(* Logix 5000 project; controller cal1632 1756-L62 rev 16.20; software revision 16.05; part 7 of 61 *)
(* tags used below, declared in another part *)
   tmrFlash : TIMER[4];   // Flash Timer
   aaa_aaa_temp : BOOL;
   FAULT : BOOL;
   FlashBit_500MSec : BOOL;   // Flash Bit 500 MSec
   p00_FlashBit_1Sec : BOOL;   // System Flash Bit 1 Second
   p00_wac : Accumulator;   // Winder Accumulator
   p01_int_from_oxidizer : INT[10];
   p01_param_master_accel : REAL;
   p01_param_master_decel : REAL;
   p01_param_master_jog_accel : REAL;
   p01_param_master_jog_decel : REAL;
   p01_param_master_jog_speed : REAL;
   p01_param_oven_timer_presets : DINT[32];
   p01_param_slow_speed_sp : REAL;
   p01_param_start_delay : REAL;
   p01_param_tension_deviation : REAL;
   p01_recipe_active : recipe;
   p01r01 : routine;
   p01r02_do_buzzer : BOOL;
   p01r02_do_buzzer_LINE : BOOL;
   p01r02_do_green_stack_light_lel : BOOL;
   p01r02_do_green_stack_light_LINE : BOOL;
   p01r02_do_horn : BOOL;
   p01r02_do_red_stack_light : BOOL;
   p01r02_do_red_stack_light_LINE : BOOL;
   p01r02_do_yellow_stack_light : BOOL;
   p01r02_do_yellow_stack_light_LINE : BOOL;
   p01r02_plc_scan_time_in_sec : REAL;
   p01r02_timer_second : TIMER[2];
   p01r09 : routine;
   p01r09_mode_run : BOOL;
   p01r09_open_oven : BOOL;
   p01r09_pb_global_reset : BOOL;
   p01r09_pb_line_jog : BOOL;
   p01r09_request_line_jog : BOOL;
   p01r10 : routine;
   p01r10_timer_fault : TIMER[4];
   p01r10_timer_warning : TIMER[4];
   p01r10_unack_fault_ex : BOOL;
   p01r10_unack_warn_ex : BOOL;
   p01r11 : routine;
   p01r11_timer_fault : TIMER[4];
   p01r11_timer_warning : TIMER[4];
   p01r12 : routine;
   p01r12_accel_rate : REAL;
   p01r12_decel_rate : REAL;
   p01r12_line_at_speed : BOOL;
   p01r12_master_acel_decel_ramp : SYS_ACC_DEC_RAMP;
   p01r12_master_ramped_speed : REAL;
   p01r12_ramped_setpoint : REAL;
   p01r12_request_any_jog_thread : BOOL;
   p01r12_selected_line_speed : REAL;
   p01r12_timer_fault : TIMER[8];
   p01r12_timer_warning : TIMER[8];
   p01r12_zero_line_speed : BOOL;
   p01r13 : routine;
   p01r13_check_status : BOOL;
   p01r13_check_status_time : REAL;
   p01r13_check_status_timer : TIMER;
   p01r13_check_tension : TIMER;
   p01r13_letoff_tension_ok : BOOL;
   p01r13_LFL_stop : BOOL;
   p01r13_line_running : BOOL;
   p01r13_line_slow_ramp : BOOL;
   p01r13_line_start : SYS_ENC;
   p01r13_oven_temp_ok : BOOL;
   p01r13_pb_start : BOOL;
   p01r13_pb_stop : BOOL;
   p01r13_permissive_drives : BOOL;
   p01r13_permissive_line_run : BOOL;
   p01r13_permissive_oven : BOOL;
   p01r13_permissive_oxidizer : BOOL;
   p01r13_request_run : BOOL;
   p01r13_request_stop : BOOL;
   p01r13_state : DINT;
   p01r13_status : DINT;
   p01r13_system_mode_run : BOOL;
   p01r13_temperature_status_check : TIMER;
   p01r13_tension_ok : BOOL;
   p01r13_timer_line_start_warning_dwell : TIMER;
   p01r13_timer_line_stop_dwell : TIMER;
   p01r13_timer_switch_to_stretch_dwell : TIMER;
   p01r13_ts1_tension_ok : BOOL;
   p01r13_ts2_tension_ok : BOOL;
   p01r13_winder_tension_ok : BOOL;
   p01r14 : routine;
   p02_dint_from_hmi : hmi_dint;
   p02_real_from_hmi : hmi_real;
   p11r30 : routine;
   p11r30_request_heat : BOOL;
   p11r31 : routine;
   p12r30 : routine;
   p12r30_request_heat : BOOL;
   p12r31 : routine;
   p13r30 : routine;
   p13r30_request_cool : BOOL;
   p20_di_acc_empty : BOOL;
   p20_do_close_nip : BOOL;
   p20r02_letoff_selection_dwell : TIMER;
   p20r10 : routine;
   p20r10_pid_tens : PID;
   p20r15 : routine;
   p20r15_loa_on : BOOL;
   p20r16 : routine;
   p20r16_lob_on : BOOL;
   p20r18_index_complete : BOOL;
   p22_param_ts1_jog_speed : REAL;
   p22r09_mode_run : BOOL;
   p22r09_mode_thread : BOOL;
   p22r09_pb_jog_fwd : BOOL;
   p22r09_pb_jog_rev : BOOL;
   p22r10_pid_psn : PID;
   p22r11 : routine;
   p22r11_request_thread_fwd : BOOL;
   p22r11_request_thread_rev : BOOL;
   p23_di_impreg_tank_up : BOOL;
   p23_param_mtr_jog_speed : REAL;
   p23r02 : routine;
   p23r15 : routine;
   p25_param_ts2_jog_speed : REAL;
   p25r09_mode_run : BOOL;
   p25r09_mode_thread : BOOL;
   p25r09_pb_jog_fwd : BOOL;
   p25r09_pb_jog_rev : BOOL;
   p25r10_pid_psn : PID;
   p25r11 : routine;
   p25r11_request_thread_fwd : BOOL;
   p25r11_request_thread_rev : BOOL;
   p28r11 : routine;
   p29_param_winder_jog_speed : REAL;
   p29r02_winder_selection_dwell : TIMER;
   p29r10_tension_error : REAL;   // Winder Winder A Tension Error winder_tension_sp - Load Cell [lbf]
   p29r11_line_start : BOOL;
   p29r11_line_stop : BOOL;
   p29r15 : routine;
   p29r15_wdra_active : BOOL;
   p29r16 : routine;
   p29r16_wdrb_active : BOOL;
   p31r09 : routine;
(* P01_System, continued *)

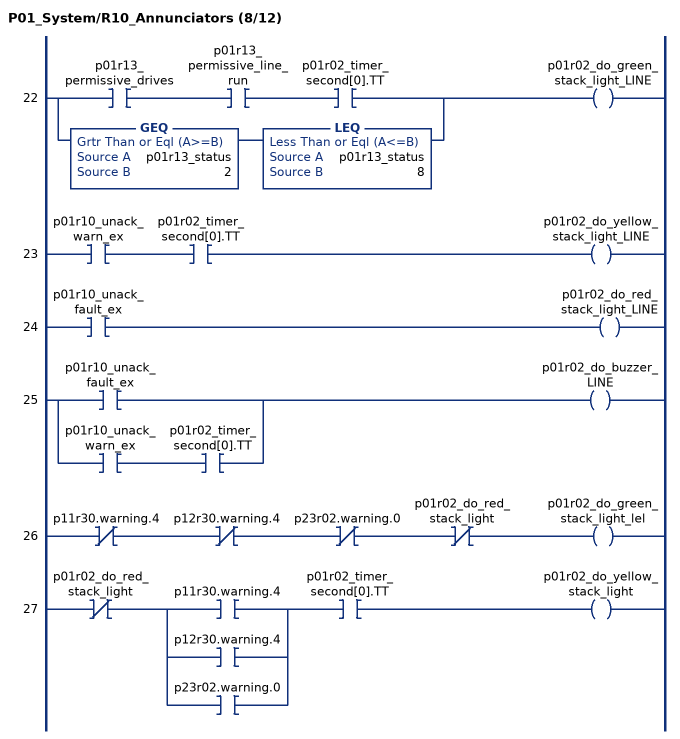
   [picture p99: P01_System/R10_Annunciators rungs 22-27]
   22: [XIC(p01r13_permissive_drives) XIC(p01r13_permissive_line_run) XIC(p01r02_timer_second[0].TT) ,GEQ(p01r13_status,2) LEQ(p01r13_status,8) ]OTE(p01r02_do_green_stack_light_LINE);
   23: XIC(p01r10_unack_warn_ex)XIC(p01r02_timer_second[0].TT)OTE(p01r02_do_yellow_stack_light_LINE);
   24: XIC(p01r10_unack_fault_ex)OTE(p01r02_do_red_stack_light_LINE);
   25: [XIC(p01r10_unack_fault_ex) ,XIC(p01r10_unack_warn_ex) XIC(p01r02_timer_second[0].TT) ]OTE(p01r02_do_buzzer_LINE);
   26: XIO(p11r30.warning.4)XIO(p12r30.warning.4)XIO(p23r02.warning.0)XIO(p01r02_do_red_stack_light)OTE(p01r02_do_green_stack_light_lel);
   27: XIO(p01r02_do_red_stack_light)[XIC(p11r30.warning.4) ,XIC(p12r30.warning.4) ,XIC(p23r02.warning.0) ]XIC(p01r02_timer_second[0].TT)OTE(p01r02_do_yellow_stack_light);
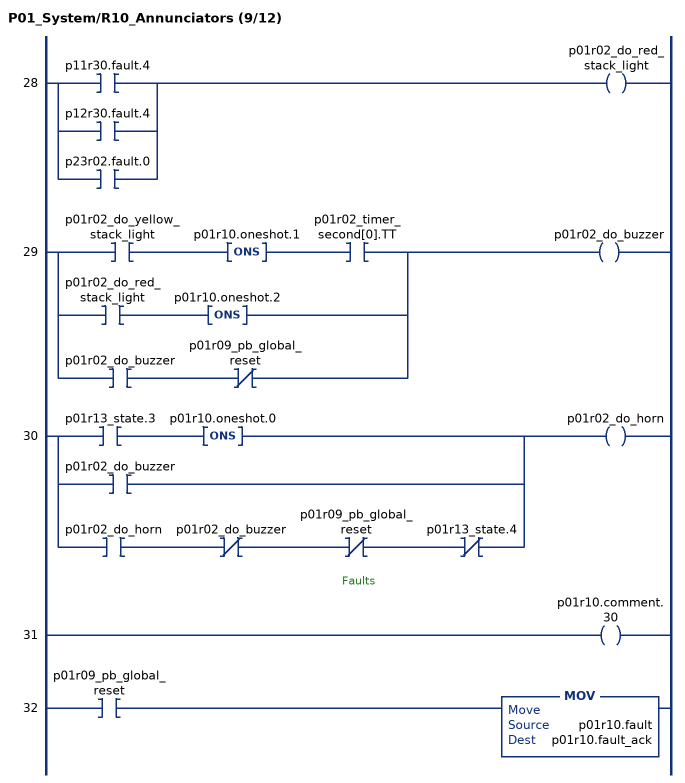
   28: [XIC(p11r30.fault.4) ,XIC(p12r30.fault.4) ,XIC(p23r02.fault.0) ]OTE(p01r02_do_red_stack_light);
   29: [[XIC(p01r02_do_yellow_stack_light) ONS(p01r10.oneshot.1) XIC(p01r02_timer_second[0].TT) ,XIC(p01r02_do_red_stack_light) ONS(p01r10.oneshot.2) ] ,XIC(p01r02_do_buzzer) XIO(p01r09_pb_global_reset) ]OTE(p01r02_do_buzzer);
   30: [[XIC(p01r13_state.3) ONS(p01r10.oneshot.0) ,XIC(p01r02_do_buzzer) ] ,XIC(p01r02_do_horn) XIO(p01r02_do_buzzer) XIO(p01r09_pb_global_reset) XIO(p01r13_state.4) ]OTE(p01r02_do_horn);
   // Faults
   31: OTE(p01r10.comment.30);
   32: XIC(p01r09_pb_global_reset)MOV(p01r10.fault,p01r10.fault_ack);
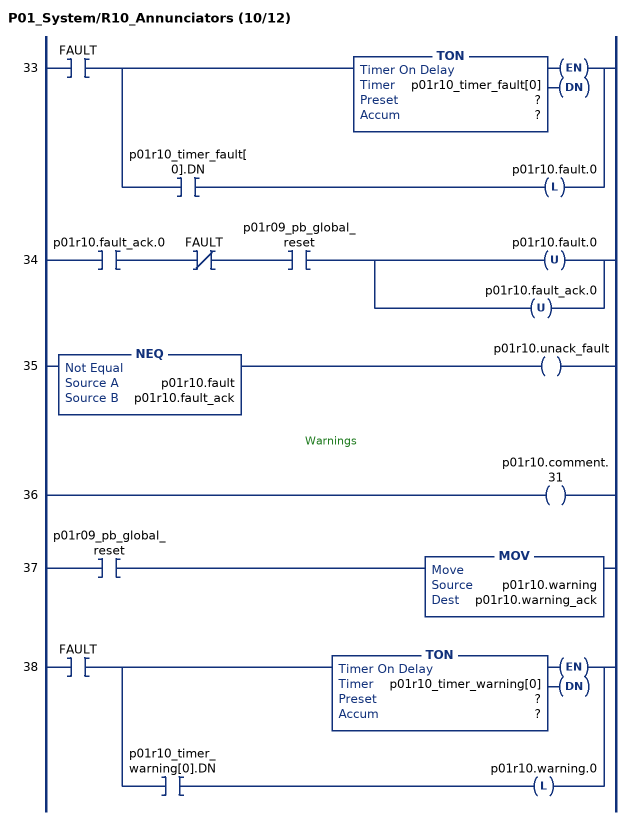
   33: XIC(FAULT)[TON(p01r10_timer_fault[0],?,?) ,XIC(p01r10_timer_fault[0].DN) OTL(p01r10.fault.0) ];
   34: XIC(p01r10.fault_ack.0)XIO(FAULT)XIC(p01r09_pb_global_reset)[OTU(p01r10.fault.0) ,OTU(p01r10.fault_ack.0) ];
   35: NEQ(p01r10.fault,p01r10.fault_ack)OTE(p01r10.unack_fault);
   // Warnings
   36: OTE(p01r10.comment.31);
   37: XIC(p01r09_pb_global_reset)MOV(p01r10.warning,p01r10.warning_ack);
   38: XIC(FAULT)[TON(p01r10_timer_warning[0],?,?) ,XIC(p01r10_timer_warning[0].DN) OTL(p01r10.warning.0) ];
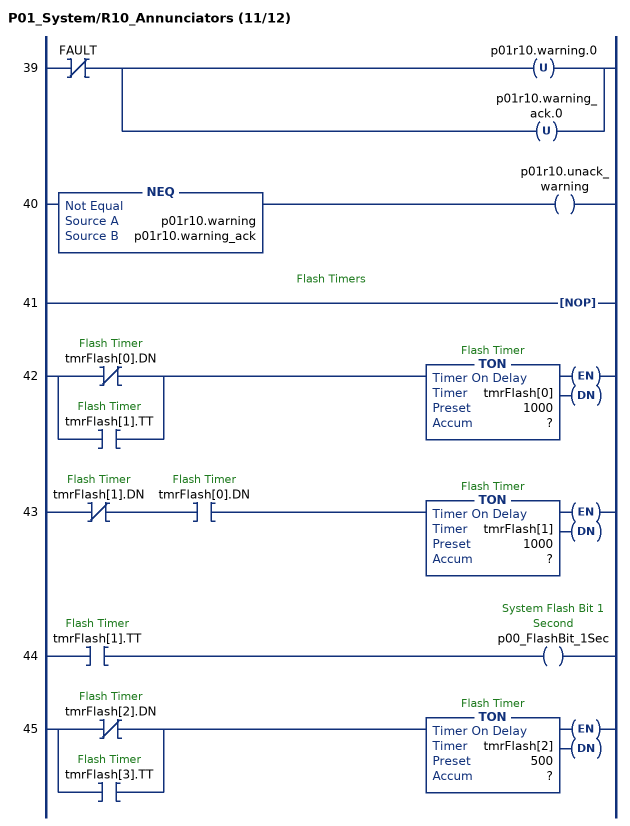
   39: XIO(FAULT)[OTU(p01r10.warning.0) ,OTU(p01r10.warning_ack.0) ];
   40: NEQ(p01r10.warning,p01r10.warning_ack)OTE(p01r10.unack_warning);
   // Flash Timers
   41: NOP();
   42: [XIO(tmrFlash[0].DN) ,XIC(tmrFlash[1].TT) ]TON(tmrFlash[0],?,?);
   43: XIO(tmrFlash[1].DN)XIC(tmrFlash[0].DN)TON(tmrFlash[1],?,?);
   44: XIC(tmrFlash[1].TT)OTE(p00_FlashBit_1Sec);
   45: [XIO(tmrFlash[2].DN) ,XIC(tmrFlash[3].TT) ]TON(tmrFlash[2],?,?);
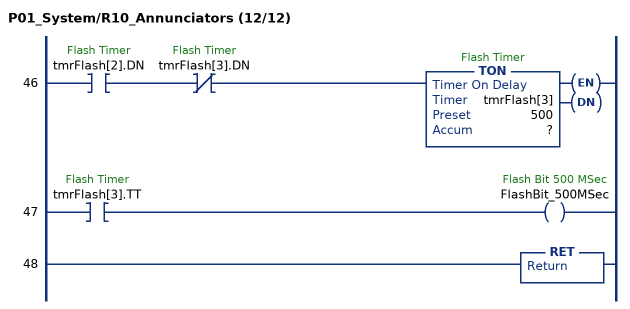
   46: XIC(tmrFlash[2].DN)XIO(tmrFlash[3].DN)TON(tmrFlash[3],?,?);
   47: XIC(tmrFlash[3].TT)OTE(FlashBit_500MSec);
   48: RET();
END_ROUTINE

ROUTINE R11_Oven_Timer_Presets   (* ladder *)
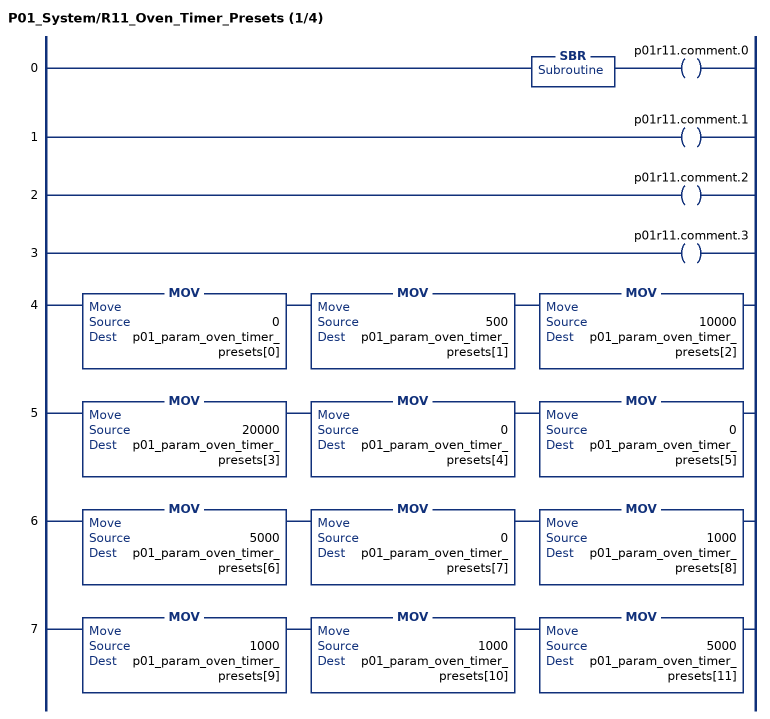
   0: SBR()OTE(p01r11.comment.0);
   1: OTE(p01r11.comment.1);
   2: OTE(p01r11.comment.2);
   3: OTE(p01r11.comment.3);
   4: MOV(0,p01_param_oven_timer_presets[0])MOV(500,p01_param_oven_timer_presets[1])MOV(10000,p01_param_oven_timer_presets[2]);
   5: MOV(20000,p01_param_oven_timer_presets[3])MOV(0,p01_param_oven_timer_presets[4])MOV(0,p01_param_oven_timer_presets[5]);
   6: MOV(5000,p01_param_oven_timer_presets[6])MOV(0,p01_param_oven_timer_presets[7])MOV(1000,p01_param_oven_timer_presets[8]);
   7: MOV(1000,p01_param_oven_timer_presets[9])MOV(1000,p01_param_oven_timer_presets[10])MOV(5000,p01_param_oven_timer_presets[11]);
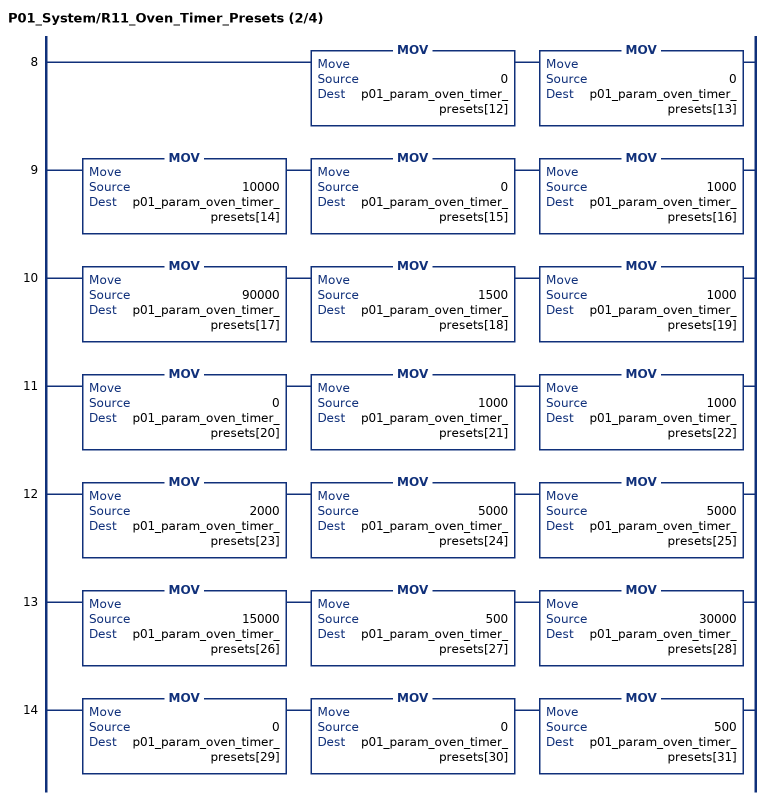
   8: MOV(0,p01_param_oven_timer_presets[12])MOV(0,p01_param_oven_timer_presets[13]);
   9: MOV(10000,p01_param_oven_timer_presets[14])MOV(0,p01_param_oven_timer_presets[15])MOV(1000,p01_param_oven_timer_presets[16]);
   10: MOV(90000,p01_param_oven_timer_presets[17])MOV(1500,p01_param_oven_timer_presets[18])MOV(1000,p01_param_oven_timer_presets[19]);
   11: MOV(0,p01_param_oven_timer_presets[20])MOV(1000,p01_param_oven_timer_presets[21])MOV(1000,p01_param_oven_timer_presets[22]);
   12: MOV(2000,p01_param_oven_timer_presets[23])MOV(5000,p01_param_oven_timer_presets[24])MOV(5000,p01_param_oven_timer_presets[25]);
   13: MOV(15000,p01_param_oven_timer_presets[26])MOV(500,p01_param_oven_timer_presets[27])MOV(30000,p01_param_oven_timer_presets[28]);
   14: MOV(0,p01_param_oven_timer_presets[29])MOV(0,p01_param_oven_timer_presets[30])MOV(500,p01_param_oven_timer_presets[31]);
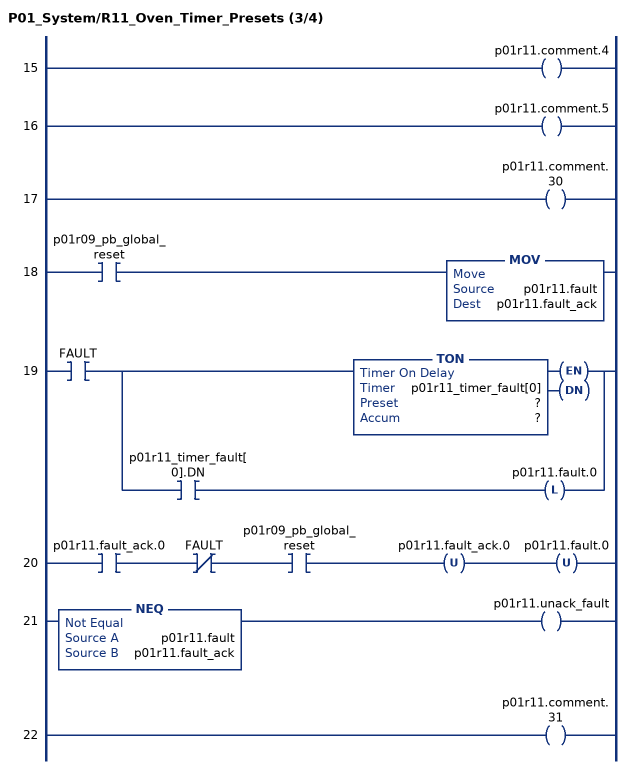
   15: OTE(p01r11.comment.4);
   16: OTE(p01r11.comment.5);
   17: OTE(p01r11.comment.30);
   18: XIC(p01r09_pb_global_reset)MOV(p01r11.fault,p01r11.fault_ack);
   19: XIC(FAULT)[TON(p01r11_timer_fault[0],?,?) ,XIC(p01r11_timer_fault[0].DN) OTL(p01r11.fault.0) ];
   20: XIC(p01r11.fault_ack.0)XIO(FAULT)XIC(p01r09_pb_global_reset)OTU(p01r11.fault_ack.0)OTU(p01r11.fault.0);
   21: NEQ(p01r11.fault,p01r11.fault_ack)OTE(p01r11.unack_fault);
   22: OTE(p01r11.comment.31);
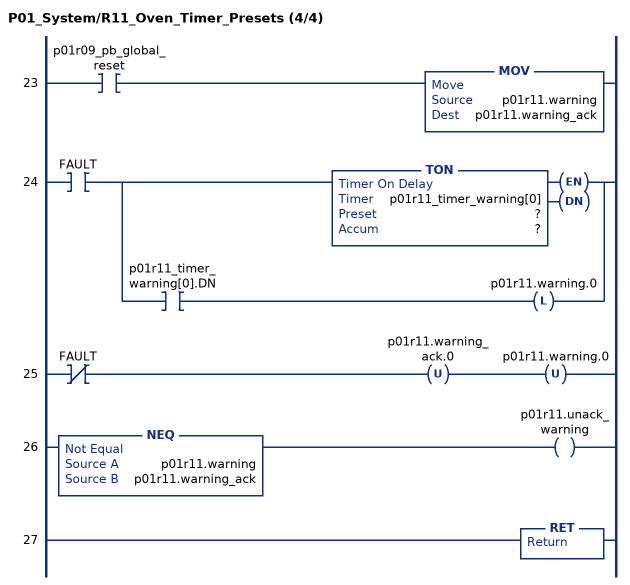
   23: XIC(p01r09_pb_global_reset)MOV(p01r11.warning,p01r11.warning_ack);
   24: XIC(FAULT)[TON(p01r11_timer_warning[0],?,?) ,XIC(p01r11_timer_warning[0].DN) OTL(p01r11.warning.0) ];
   25: XIO(FAULT)OTU(p01r11.warning_ack.0)OTU(p01r11.warning.0);
   26: NEQ(p01r11.warning,p01r11.warning_ack)OTE(p01r11.unack_warning);
   27: RET();
END_ROUTINE

ROUTINE R12_Line_Accel_Decel_Control   (* ladder *)
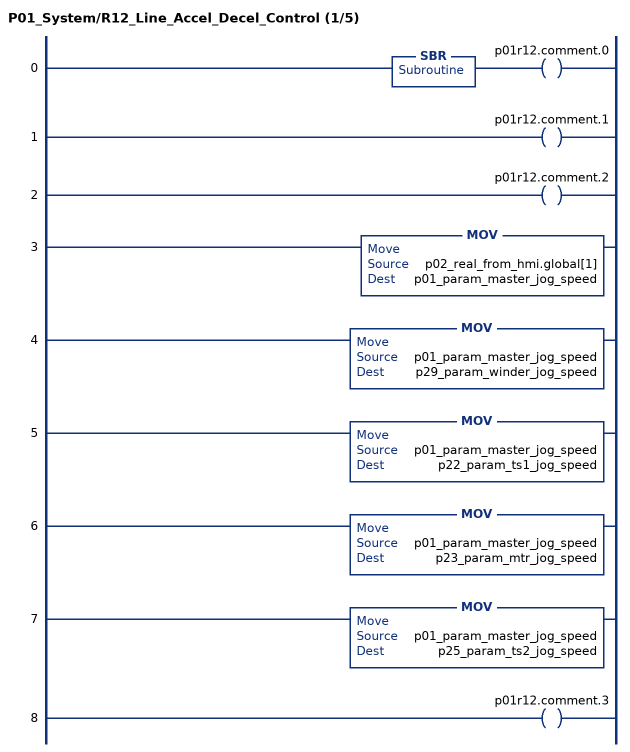
   0: SBR()OTE(p01r12.comment.0);
   1: OTE(p01r12.comment.1);
   2: OTE(p01r12.comment.2);
   3: MOV(p02_real_from_hmi.global[1],p01_param_master_jog_speed);
   4: MOV(p01_param_master_jog_speed,p29_param_winder_jog_speed);
   5: MOV(p01_param_master_jog_speed,p22_param_ts1_jog_speed);
   6: MOV(p01_param_master_jog_speed,p23_param_mtr_jog_speed);
   7: MOV(p01_param_master_jog_speed,p25_param_ts2_jog_speed);
   8: OTE(p01r12.comment.3);
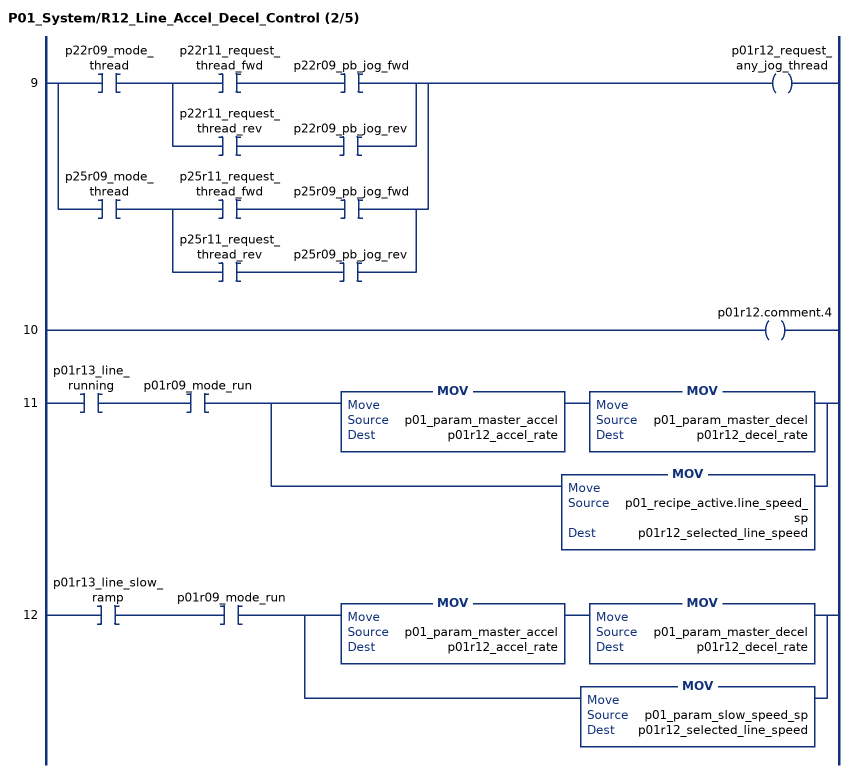
   9: [XIC(p22r09_mode_thread) [XIC(p22r11_request_thread_fwd) XIC(p22r09_pb_jog_fwd) ,XIC(p22r11_request_thread_rev) XIC(p22r09_pb_jog_rev) ] ,XIC(p25r09_mode_thread) [XIC(p25r11_request_thread_fwd) XIC(p25r09_pb_jog_fwd) ,XIC(p25r11_request_thread_rev) XIC(p25r09_pb_jog_rev) ] ]OTE(p01r12_request_any_jog_thread);
   10: OTE(p01r12.comment.4);
   11: XIC(p01r13_line_running)XIC(p01r09_mode_run)[MOV(p01_param_master_accel,p01r12_accel_rate) MOV(p01_param_master_decel,p01r12_decel_rate) ,MOV(p01_recipe_active.line_speed_sp,p01r12_selected_line_speed) ];
   12: XIC(p01r13_line_slow_ramp)XIC(p01r09_mode_run)[MOV(p01_param_master_accel,p01r12_accel_rate) MOV(p01_param_master_decel,p01r12_decel_rate) ,MOV(p01_param_slow_speed_sp,p01r12_selected_line_speed) ];
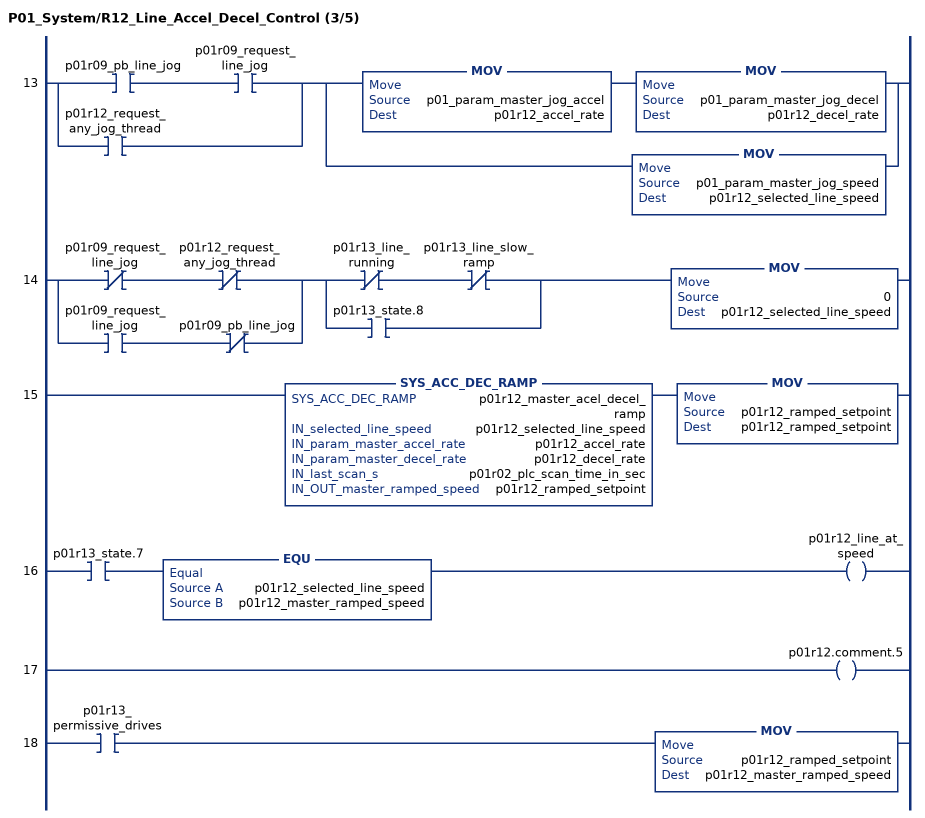
   13: [XIC(p01r09_pb_line_jog) XIC(p01r09_request_line_jog) ,XIC(p01r12_request_any_jog_thread) ][MOV(p01_param_master_jog_accel,p01r12_accel_rate) MOV(p01_param_master_jog_decel,p01r12_decel_rate) ,MOV(p01_param_master_jog_speed,p01r12_selected_line_speed) ];
   14: [XIO(p01r09_request_line_jog) XIO(p01r12_request_any_jog_thread) ,XIC(p01r09_request_line_jog) XIO(p01r09_pb_line_jog) ][XIO(p01r13_line_running) XIO(p01r13_line_slow_ramp) ,XIC(p01r13_state.8) ]MOV(0,p01r12_selected_line_speed);
   15: SYS_ACC_DEC_RAMP(p01r12_master_acel_decel_ramp,p01r12_selected_line_speed,p01r12_accel_rate,p01r12_decel_rate,p01r02_plc_scan_time_in_sec,p01r12_ramped_setpoint)MOV(p01r12_ramped_setpoint,p01r12_ramped_setpoint);
   16: XIC(p01r13_state.7)EQU(p01r12_selected_line_speed,p01r12_master_ramped_speed)OTE(p01r12_line_at_speed);
   17: OTE(p01r12.comment.5);
   18: XIC(p01r13_permissive_drives)MOV(p01r12_ramped_setpoint,p01r12_master_ramped_speed);
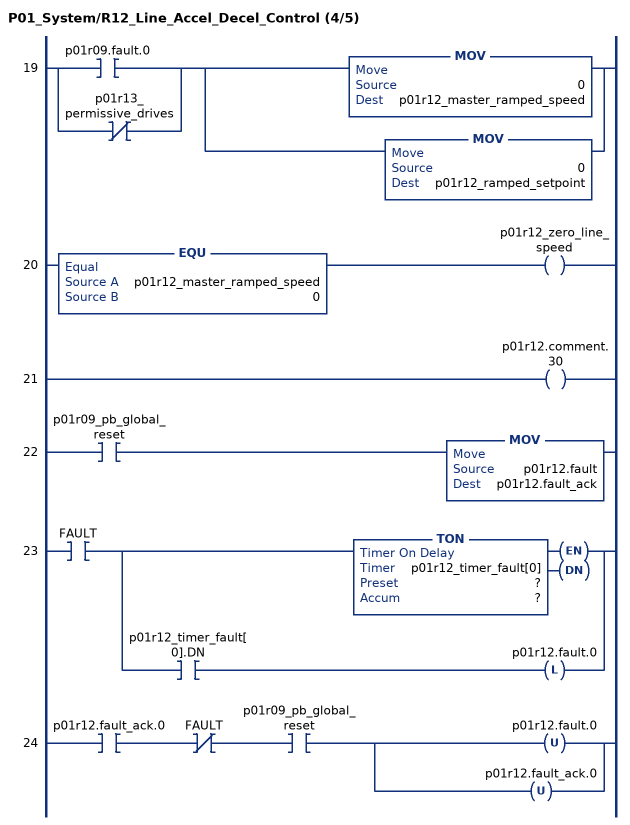
   19: [XIC(p01r09.fault.0) ,XIO(p01r13_permissive_drives) ][MOV(0,p01r12_master_ramped_speed) ,MOV(0,p01r12_ramped_setpoint) ];
   20: EQU(p01r12_master_ramped_speed,0)OTE(p01r12_zero_line_speed);
   21: OTE(p01r12.comment.30);
   22: XIC(p01r09_pb_global_reset)MOV(p01r12.fault,p01r12.fault_ack);
   23: XIC(FAULT)[TON(p01r12_timer_fault[0],?,?) ,XIC(p01r12_timer_fault[0].DN) OTL(p01r12.fault.0) ];
   24: XIC(p01r12.fault_ack.0)XIO(FAULT)XIC(p01r09_pb_global_reset)[OTU(p01r12.fault.0) ,OTU(p01r12.fault_ack.0) ];
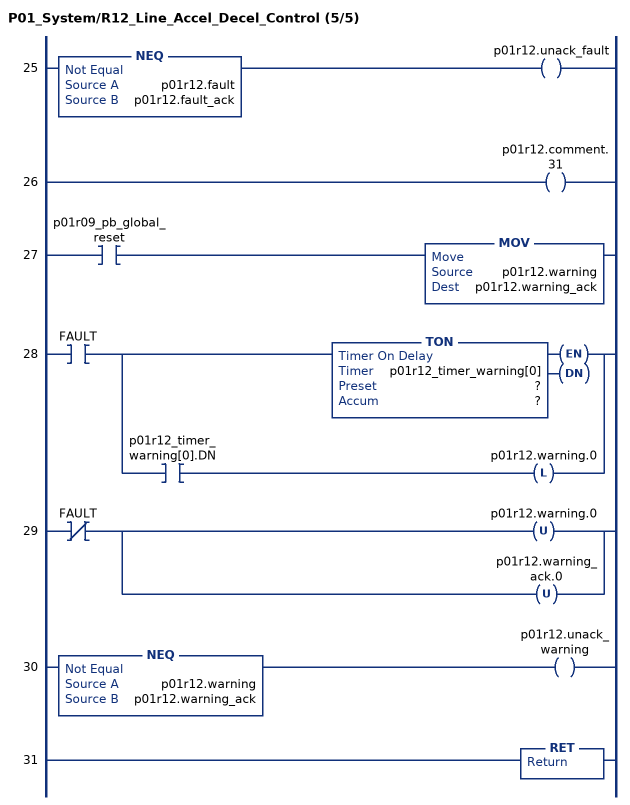
   25: NEQ(p01r12.fault,p01r12.fault_ack)OTE(p01r12.unack_fault);
   26: OTE(p01r12.comment.31);
   27: XIC(p01r09_pb_global_reset)MOV(p01r12.warning,p01r12.warning_ack);
   28: XIC(FAULT)[TON(p01r12_timer_warning[0],?,?) ,XIC(p01r12_timer_warning[0].DN) OTL(p01r12.warning.0) ];
   29: XIO(FAULT)[OTU(p01r12.warning.0) ,OTU(p01r12.warning_ack.0) ];
   30: NEQ(p01r12.warning,p01r12.warning_ack)OTE(p01r12.unack_warning);
   31: RET();
END_ROUTINE

ROUTINE R13_Line_Start_Sequence   (* ladder *)
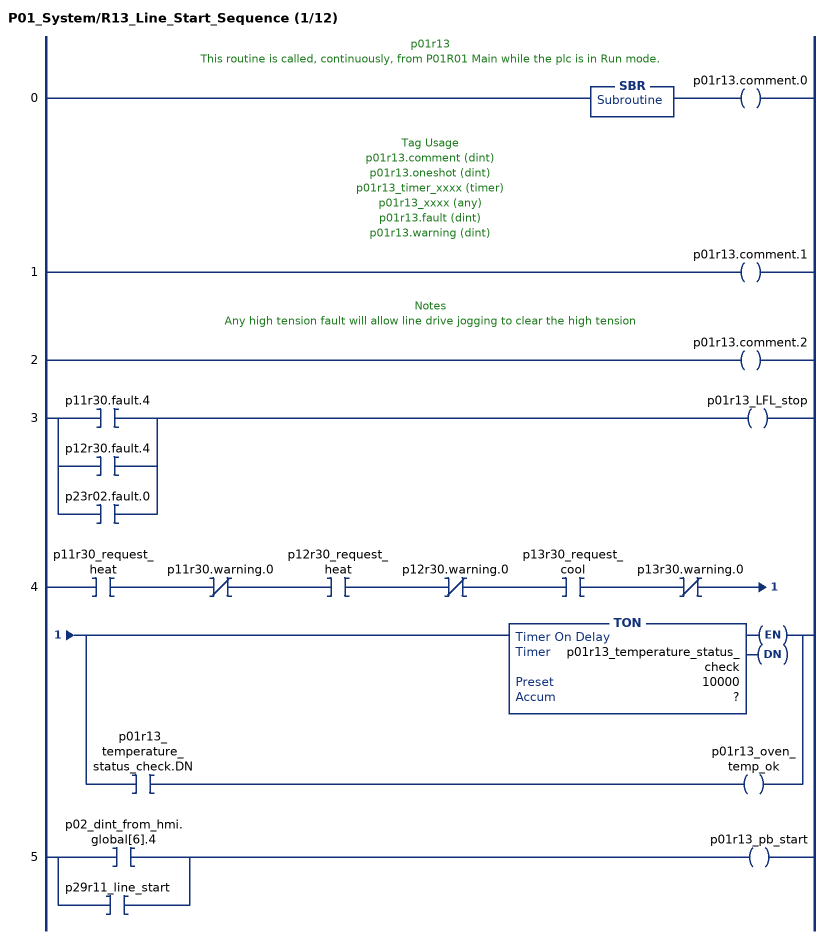
   // p01r13
   // This routine is called, continuously, from P01R01 Main while the plc is in Run mode.
   0: SBR()OTE(p01r13.comment.0);
   // Tag Usage
   // p01r13.comment (dint)
   // p01r13.oneshot (dint)
   // p01r13_timer_xxxx (timer)
   // p01r13_xxxx (any)
   // p01r13.fault (dint)
   // p01r13.warning (dint)
   1: OTE(p01r13.comment.1);
   // Notes
   // Any high tension fault will allow line drive jogging to clear the high tension
   2: OTE(p01r13.comment.2);
   3: [XIC(p11r30.fault.4) ,XIC(p12r30.fault.4) ,XIC(p23r02.fault.0) ]OTE(p01r13_LFL_stop);
   4: XIC(p11r30_request_heat)XIO(p11r30.warning.0)XIC(p12r30_request_heat)XIO(p12r30.warning.0)XIC(p13r30_request_cool)XIO(p13r30.warning.0)[TON(p01r13_temperature_status_check,?,?) ,XIC(p01r13_temperature_status_check.DN) OTE(p01r13_oven_temp_ok) ];
   5: [XIC(p02_dint_from_hmi.global[6].4) ,XIC(p29r11_line_start) ]OTE(p01r13_pb_start);
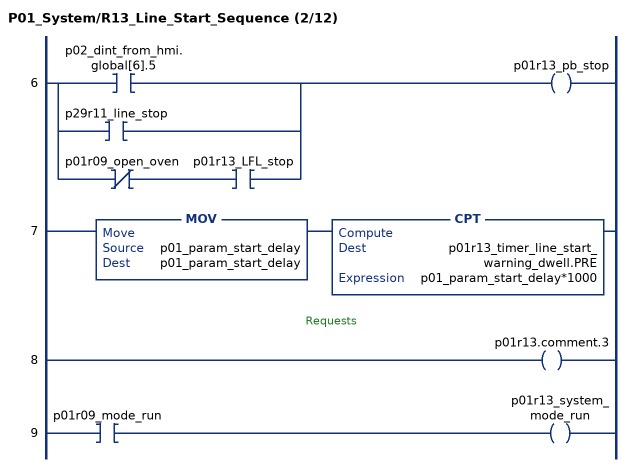
   6: [XIC(p02_dint_from_hmi.global[6].5) ,XIC(p29r11_line_stop) ,XIO(p01r09_open_oven) XIC(p01r13_LFL_stop) ]OTE(p01r13_pb_stop);
   7: MOV(p01_param_start_delay,p01_param_start_delay)CPT(p01r13_timer_line_start_warning_dwell.PRE,p01_param_start_delay*1000);
   // Requests
   8: OTE(p01r13.comment.3);
   9: XIC(p01r09_mode_run)OTE(p01r13_system_mode_run);
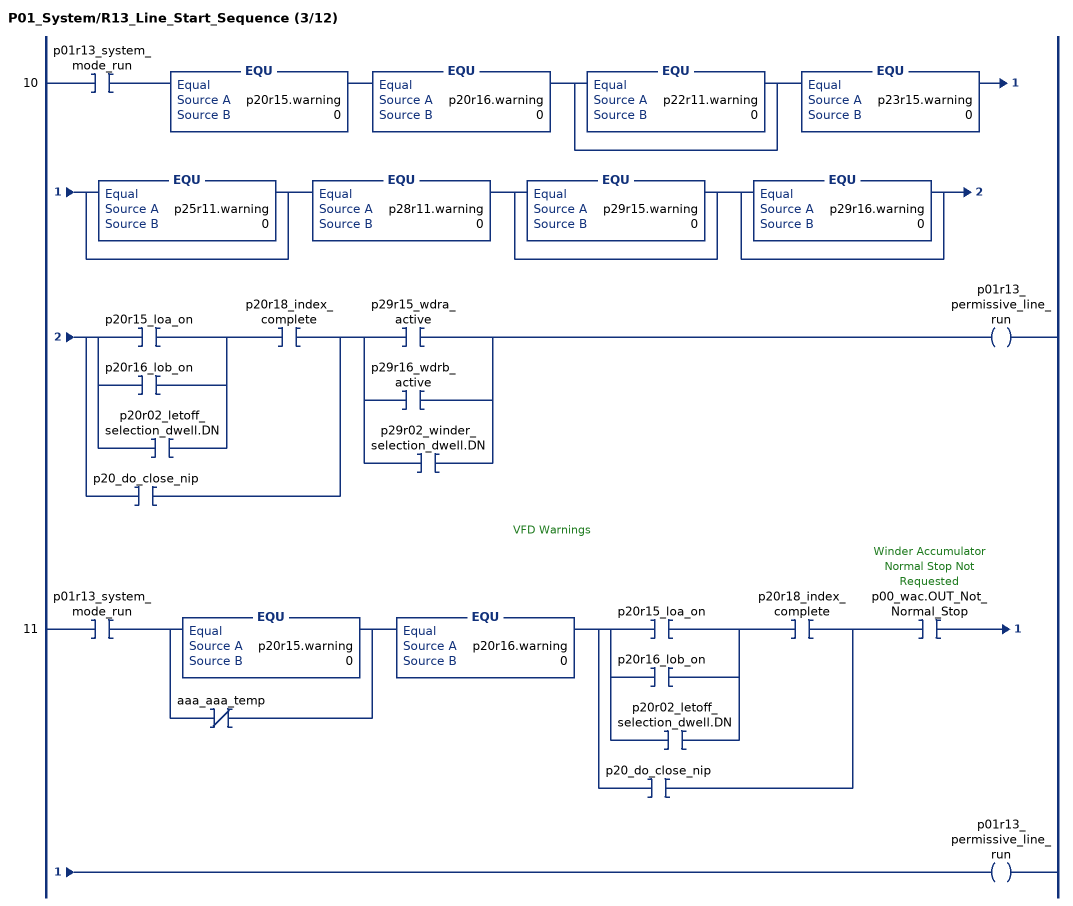
   10: XIC(p01r13_system_mode_run)EQU(p20r15.warning,0)EQU(p20r16.warning,0)[EQU(p22r11.warning,0) ,]EQU(p23r15.warning,0)[EQU(p25r11.warning,0) ,]EQU(p28r11.warning,0)[EQU(p29r15.warning,0) ,][EQU(p29r16.warning,0) ,][[XIC(p20r15_loa_on) ,XIC(p20r16_lob_on) ,XIC(p20r02_letoff_selection_dwell.DN) ] XIC(p20r18_index_complete) ,XIC(p20_do_close_nip) ][XIC(p29r15_wdra_active) ,XIC(p29r16_wdrb_active) ,XIC(p29r02_winder_selection_dwell.DN) ]OTE(p01r13_permissive_line_run);
   // VFD Warnings
   11: XIC(p01r13_system_mode_run)[EQU(p20r15.warning,0) ,XIO(aaa_aaa_temp) ]EQU(p20r16.warning,0)[[XIC(p20r15_loa_on) ,XIC(p20r16_lob_on) ,XIC(p20r02_letoff_selection_dwell.DN) ] XIC(p20r18_index_complete) ,XIC(p20_do_close_nip) ]XIC(p00_wac.OUT_Not_Normal_Stop)OTE(p01r13_permissive_line_run);
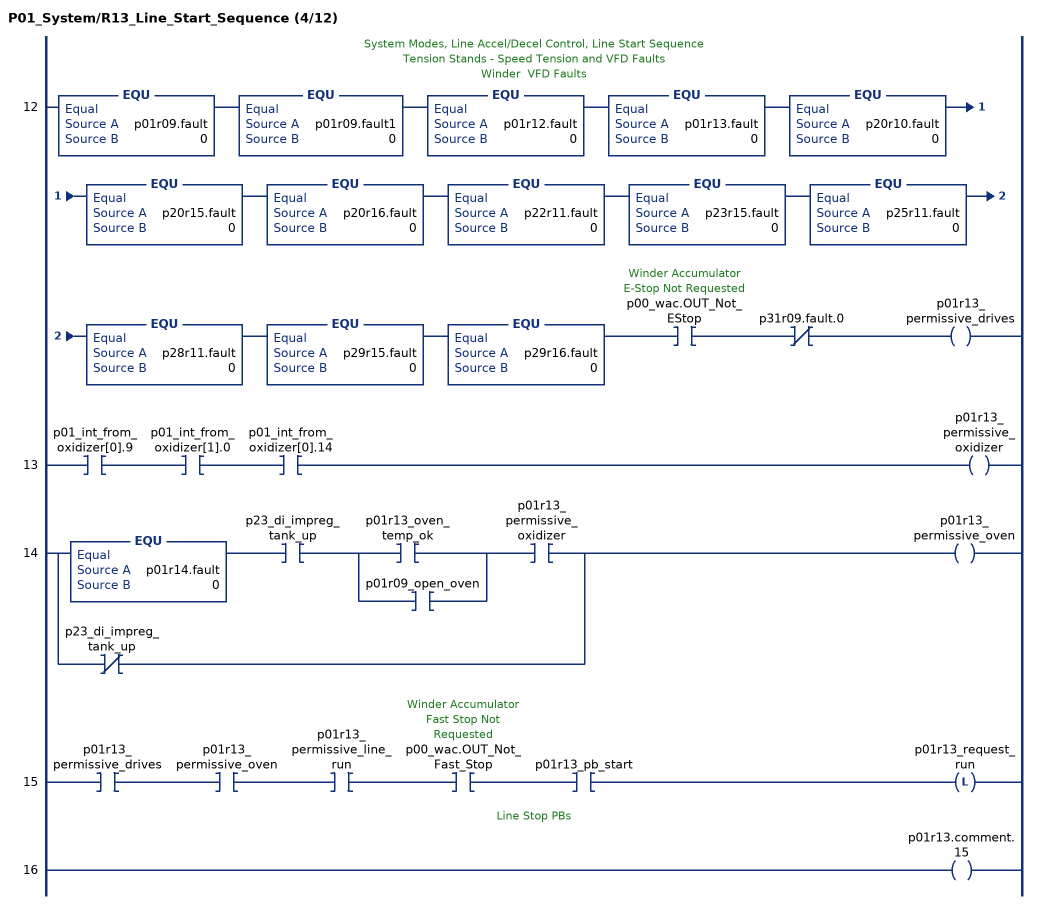
   // System Modes, Line Accel/Decel Control, Line Start Sequence
   // Tension Stands - Speed Tension and VFD Faults
   // Winder  VFD Faults
   12: EQU(p01r09.fault,0)EQU(p01r09.fault1,0)EQU(p01r12.fault,0)EQU(p01r13.fault,0)EQU(p20r10.fault,0)EQU(p20r15.fault,0)EQU(p20r16.fault,0)EQU(p22r11.fault,0)EQU(p23r15.fault,0)EQU(p25r11.fault,0)EQU(p28r11.fault,0)EQU(p29r15.fault,0)EQU(p29r16.fault,0)XIC(p00_wac.OUT_Not_EStop)XIO(p31r09.fault.0)OTE(p01r13_permissive_drives);
   13: XIC(p01_int_from_oxidizer[0].9)XIC(p01_int_from_oxidizer[1].0)XIC(p01_int_from_oxidizer[0].14)OTE(p01r13_permissive_oxidizer);
   14: [EQU(p01r14.fault,0) XIC(p23_di_impreg_tank_up) [XIC(p01r13_oven_temp_ok) ,XIC(p01r09_open_oven) ] XIC(p01r13_permissive_oxidizer) ,XIO(p23_di_impreg_tank_up) ]OTE(p01r13_permissive_oven);
   15: XIC(p01r13_permissive_drives)XIC(p01r13_permissive_oven)XIC(p01r13_permissive_line_run)XIC(p00_wac.OUT_Not_Fast_Stop)XIC(p01r13_pb_start)OTL(p01r13_request_run);
   // Line Stop PBs
   16: OTE(p01r13.comment.15);
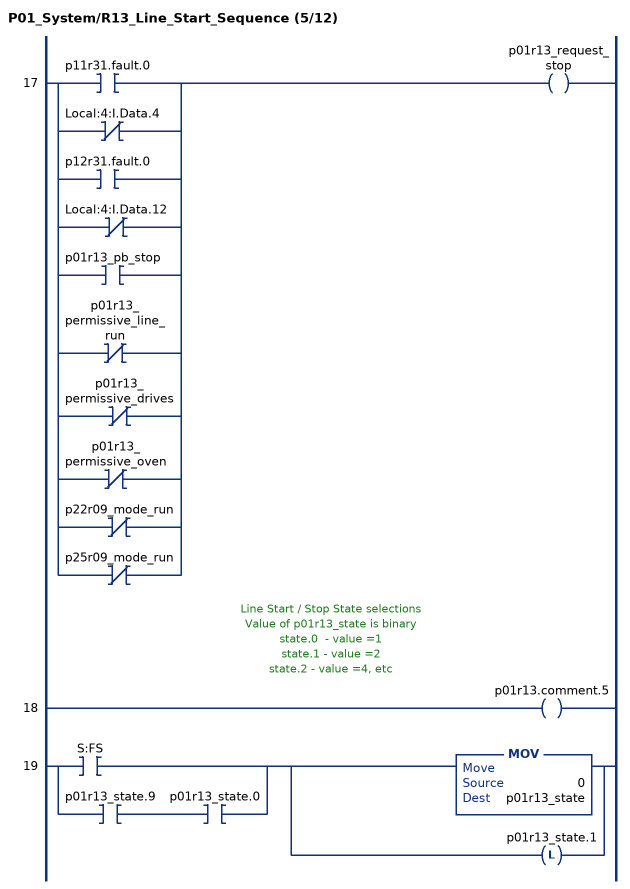
   17: [XIC(p11r31.fault.0) ,XIO(Local:4:I.Data.4) ,XIC(p12r31.fault.0) ,XIO(Local:4:I.Data.12) ,XIC(p01r13_pb_stop) ,XIO(p01r13_permissive_line_run) ,XIO(p01r13_permissive_drives) ,XIO(p01r13_permissive_oven) ,XIO(p22r09_mode_run) ,XIO(p25r09_mode_run) ]OTE(p01r13_request_stop);
   // Line Start / Stop State selections
   // Value of p01r13_state is binary
   // state.0  - value =1
   // state.1 - value =2
   // state.2 - value =4, etc
   18: OTE(p01r13.comment.5);
   19: [XIC(S:FS) ,XIC(p01r13_state.9) XIC(p01r13_state.0) ][MOV(0,p01r13_state) ,OTL(p01r13_state.1) ];
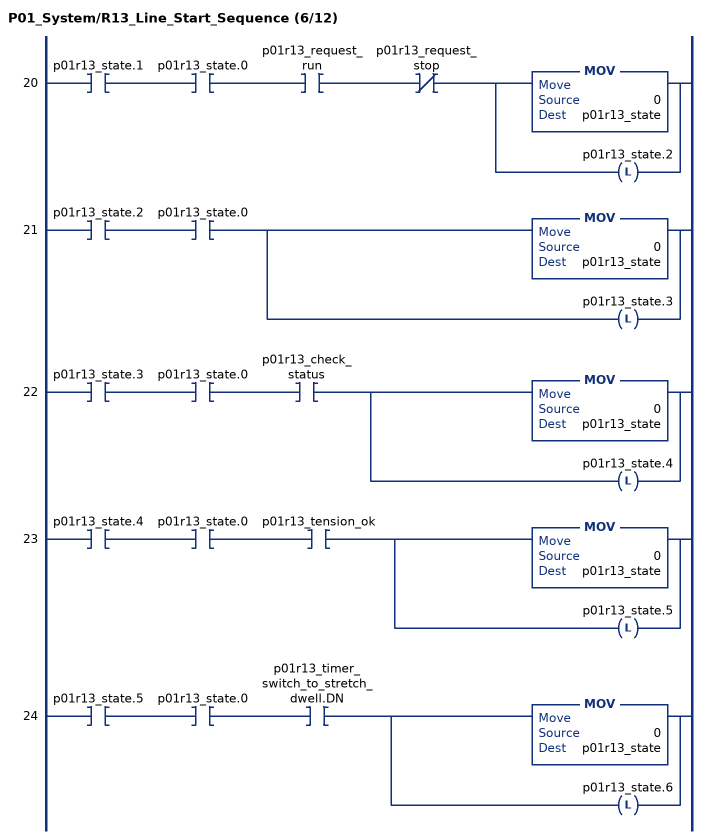
   20: XIC(p01r13_state.1)XIC(p01r13_state.0)XIC(p01r13_request_run)XIO(p01r13_request_stop)[MOV(0,p01r13_state) ,OTL(p01r13_state.2) ];
   21: XIC(p01r13_state.2)XIC(p01r13_state.0)[MOV(0,p01r13_state) ,OTL(p01r13_state.3) ];
   22: XIC(p01r13_state.3)XIC(p01r13_state.0)XIC(p01r13_check_status)[MOV(0,p01r13_state) ,OTL(p01r13_state.4) ];
   23: XIC(p01r13_state.4)XIC(p01r13_state.0)XIC(p01r13_tension_ok)[MOV(0,p01r13_state) ,OTL(p01r13_state.5) ];
   24: XIC(p01r13_state.5)XIC(p01r13_state.0)XIC(p01r13_timer_switch_to_stretch_dwell.DN)[MOV(0,p01r13_state) ,OTL(p01r13_state.6) ];
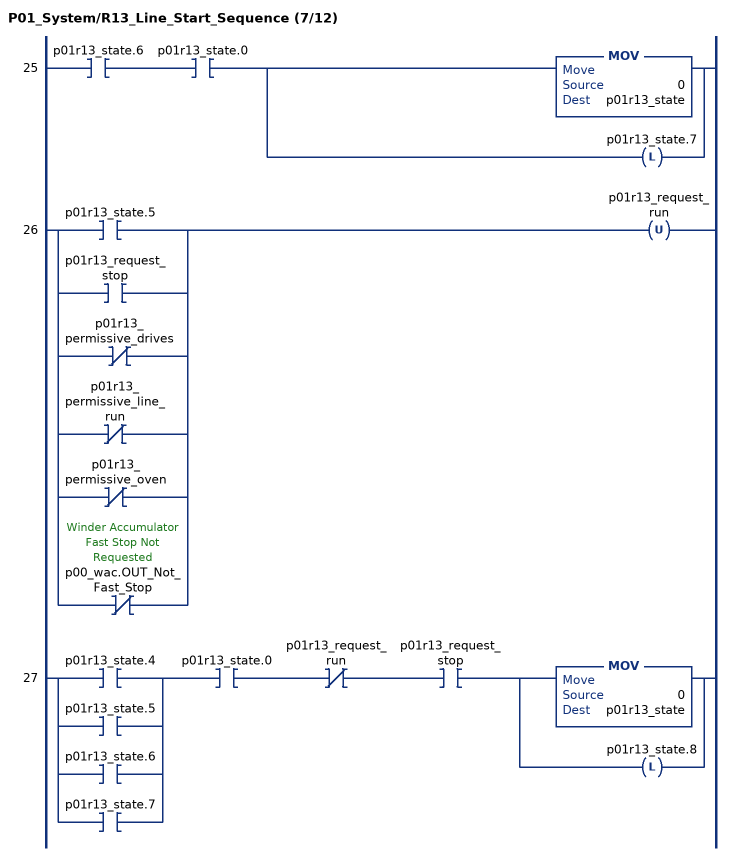
   25: XIC(p01r13_state.6)XIC(p01r13_state.0)[MOV(0,p01r13_state) ,OTL(p01r13_state.7) ];
   26: [XIC(p01r13_state.5) ,XIC(p01r13_request_stop) ,XIO(p01r13_permissive_drives) ,XIO(p01r13_permissive_line_run) ,XIO(p01r13_permissive_oven) ,XIO(p00_wac.OUT_Not_Fast_Stop) ]OTU(p01r13_request_run);
   27: [XIC(p01r13_state.4) ,XIC(p01r13_state.5) ,XIC(p01r13_state.6) ,XIC(p01r13_state.7) ]XIC(p01r13_state.0)XIO(p01r13_request_run)XIC(p01r13_request_stop)[MOV(0,p01r13_state) ,OTL(p01r13_state.8) ];
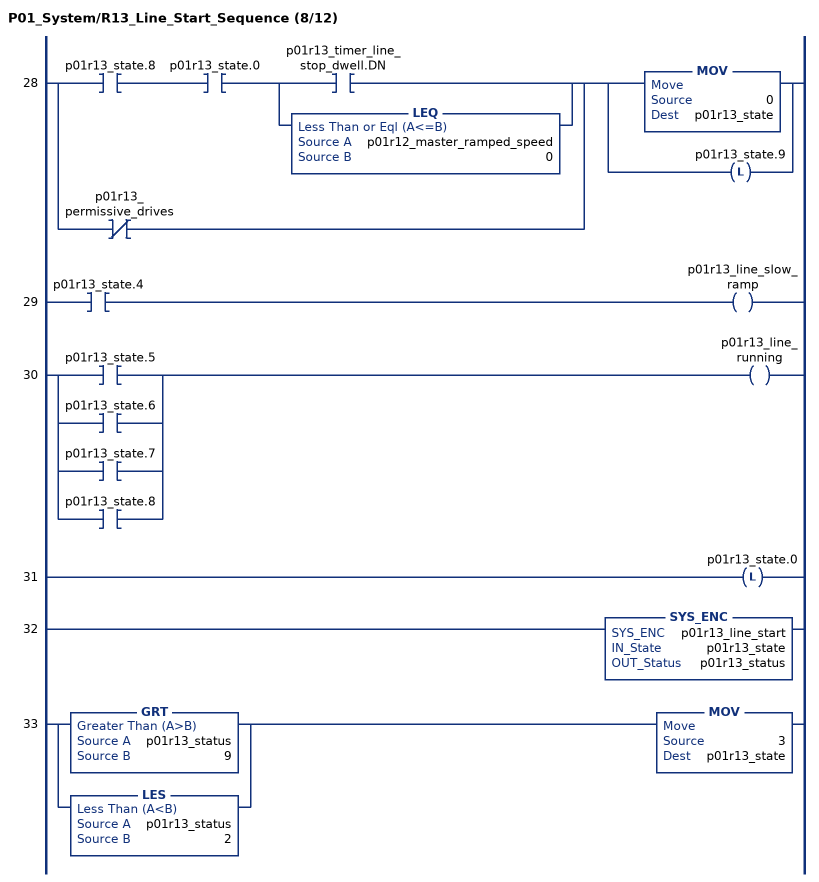
   28: [XIC(p01r13_state.8) XIC(p01r13_state.0) [XIC(p01r13_timer_line_stop_dwell.DN) ,LEQ(p01r12_master_ramped_speed,0) ] ,XIO(p01r13_permissive_drives) ][MOV(0,p01r13_state) ,OTL(p01r13_state.9) ];
   29: XIC(p01r13_state.4)OTE(p01r13_line_slow_ramp);
   30: [XIC(p01r13_state.5) ,XIC(p01r13_state.6) ,XIC(p01r13_state.7) ,XIC(p01r13_state.8) ]OTE(p01r13_line_running);
   31: OTL(p01r13_state.0);
   32: SYS_ENC(p01r13_line_start,p01r13_state,p01r13_status);
   33: [GRT(p01r13_status,9) ,LES(p01r13_status,2) ]MOV(3,p01r13_state);
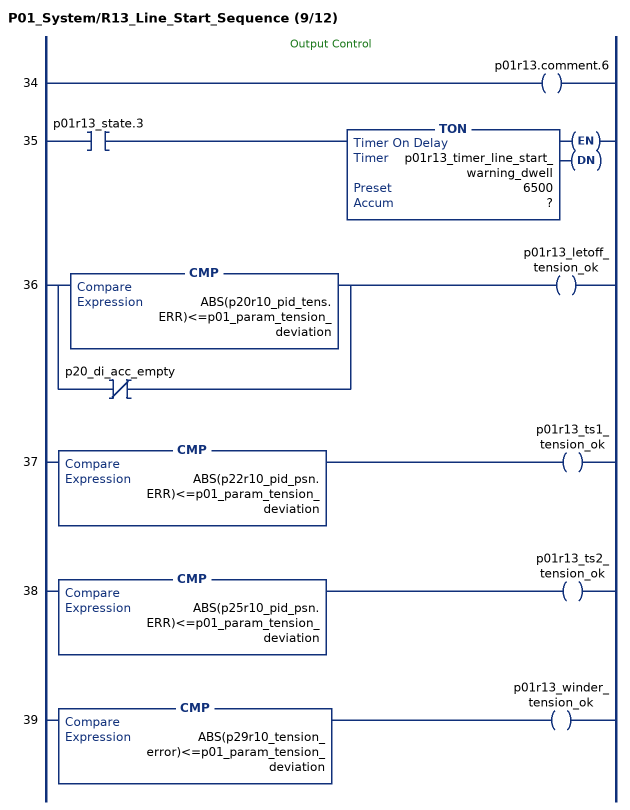
   // Output Control
   34: OTE(p01r13.comment.6);
   35: XIC(p01r13_state.3)TON(p01r13_timer_line_start_warning_dwell,?,?);
   36: [CMP(ABS(p20r10_pid_tens.ERR)<=p01_param_tension_deviation) ,XIO(p20_di_acc_empty) ]OTE(p01r13_letoff_tension_ok);
   37: CMP(ABS(p22r10_pid_psn.ERR)<=p01_param_tension_deviation)OTE(p01r13_ts1_tension_ok);
   38: CMP(ABS(p25r10_pid_psn.ERR)<=p01_param_tension_deviation)OTE(p01r13_ts2_tension_ok);
   39: CMP(ABS(p29r10_tension_error)<=p01_param_tension_deviation)OTE(p01r13_winder_tension_ok);
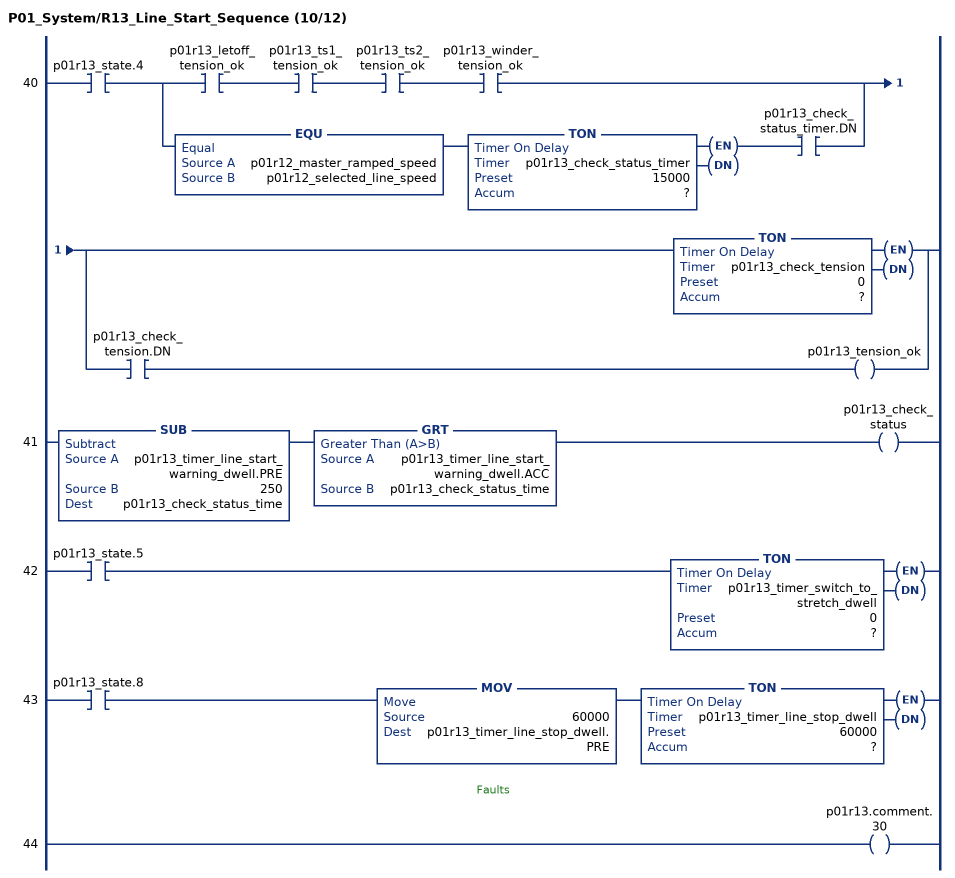
   40: XIC(p01r13_state.4)[XIC(p01r13_letoff_tension_ok) XIC(p01r13_ts1_tension_ok) XIC(p01r13_ts2_tension_ok) XIC(p01r13_winder_tension_ok) ,EQU(p01r12_master_ramped_speed,p01r12_selected_line_speed) TON(p01r13_check_status_timer,?,?) XIC(p01r13_check_status_timer.DN) ][TON(p01r13_check_tension,?,?) ,XIC(p01r13_check_tension.DN) OTE(p01r13_tension_ok) ];
   41: SUB(p01r13_timer_line_start_warning_dwell.PRE,250,p01r13_check_status_time)GRT(p01r13_timer_line_start_warning_dwell.ACC,p01r13_check_status_time)OTE(p01r13_check_status);
   42: XIC(p01r13_state.5)TON(p01r13_timer_switch_to_stretch_dwell,?,?);
   43: XIC(p01r13_state.8)MOV(60000,p01r13_timer_line_stop_dwell.PRE)TON(p01r13_timer_line_stop_dwell,?,?);
   // Faults
   44: OTE(p01r13.comment.30);
